// TIA Portal V17 export
// export: Created 2022-07-20T07:02:32.9247407Z, ExportSetting WithDefaults, DisplayName Totally Integrated Automation Portal, DisplayVersion V17, DisplayName TIA Portal Openness, DisplayVersion V17, DisplayName TIA Portal Version Control Interface, DisplayVersion V17, DisplayName SINAMICS Startdrive Advanced, DisplayVersion V17, DisplayName SINAMICS Startdrive G130, G150, S120, S150, SINAMICS MV, S210, DisplayVersion V17, DisplayName SINAMICS Startdrive G110M, G120, G120C, G120D, G120P, G115D, DisplayVersion V17, DisplayName STEP 7 Professional, DisplayVersion V17, DisplayName STEP 7 Safety, DisplayVersion V17, DisplayName WinCC Advanced, DisplayVersion V17
FUNCTION_BLOCK "FB11006_HeatingRegulation"   // FB11006, LAD
TITLE = Manage heating regulation
{ S7_Optimized_Access := 'TRUE' }
VERSION : 0.1
// stored: AutoNumber false, IsIECCheckEnabled false, IsRetainMemResEnabled false, MemoryReserve 100, SetENOAutomatically false, UDAEnableTagReadback false
   VAR_INPUT
      RequestInternalLampActivation { ExternalAccessible := 'False'; ExternalVisible := 'False'; ExternalWritable := 'False'} : Bool;
      SetpointTemperature { ExternalAccessible := 'False'; ExternalVisible := 'False'; ExternalWritable := 'False'} : Real;
      Reset { ExternalAccessible := 'False'; ExternalVisible := 'False'; ExternalWritable := 'False'} : Bool;
      TemperatureConfig { ExternalAccessible := 'False'; ExternalVisible := 'False'; ExternalWritable := 'False'} : "stTemperatureConfiguration";
      PIDConfig { ExternalAccessible := 'False'; ExternalVisible := 'False'; ExternalWritable := 'False'} : "stPIDConfiguration";
      TemperatureSensor : Int;
      ManualOptimisation : Bool;
   END_VAR
   VAR_OUTPUT
      ActiveHeating { ExternalAccessible := 'False'; ExternalVisible := 'False'; ExternalWritable := 'False'} : Bool;
      Error { ExternalAccessible := 'False'; ExternalVisible := 'False'; ExternalWritable := 'False'} : Bool;
      Alarm { ExternalAccessible := 'False'; ExternalVisible := 'False'; ExternalWritable := 'False'} : Bool;
      Warning { ExternalAccessible := 'False'; ExternalVisible := 'False'; ExternalWritable := 'False'} : Bool;
      SetPointOutput : Int;
   END_VAR
   VAR_IN_OUT
      Temperature : Real;
      PID : PID_Compact;
   END_VAR
   VAR
      R_TRIG_Enable : R_TRIG;
      F_TRIG_Enable { S7_SetPoint := 'True'} : F_TRIG;
      FB10022_Average_Instance { S7_SetPoint := 'True'} : "FB10022_Average";
      statDataAverage { S7_SetPoint := 'True'} : Array[0..29] of Real;
      statTemperatureAverage : Real;
      pid_state : Int;
      pid_error : Bool;
      pid_errorBits : DWord;
   END_VAR
   VAR_TEMP
      RET_VAL : Word;
   END_VAR
BEGIN

REGION Network 1 (SCL): Comments
   //==========================================================================================
   // SIEMENS SAS      RC-FR DI FA APC
   //------------------------------------------------------------------------------------------
   // Restrictions:    TIA V16 and more
   // Requirements:    S7-1500 + MGI library
   // Functionality:   This function block manage a PID regulation for temperature
   //------------------------------------------------------------------------------------------
   // Change log table:
   // Version      Date        Expert in charge    Changes applied
   // 01.00.01     09.06.2020  RTO                 First released version
   //==========================================================================================
END_REGION

REGION Network 2 (SCL): First Scan
   IF "FirstScan" THEN

       // Interface
       #ActiveHeating := FALSE;
       #SetPointOutput := 0;

       // #PID
       #PID.Mode := 0;
       #PID.ModeActivate := TRUE;
       #PID.IntegralResetMode := 1;

   END_IF;
END_REGION

REGION Network 3 (SCL): Edge Signal Management
   REGION EDGE SIGNALS
       #R_TRIG_Enable(CLK := #RequestInternalLampActivation);
       #F_TRIG_Enable(CLK := #RequestInternalLampActivation);

   END_REGION
END_REGION

REGION Network 4 (SCL): Convert analog input in temperature value
   #Temperature := #TemperatureConfig.ShiftFactor * #TemperatureSensor/10.0;
END_REGION

REGION Network 5: Average temperature over 30 secondes
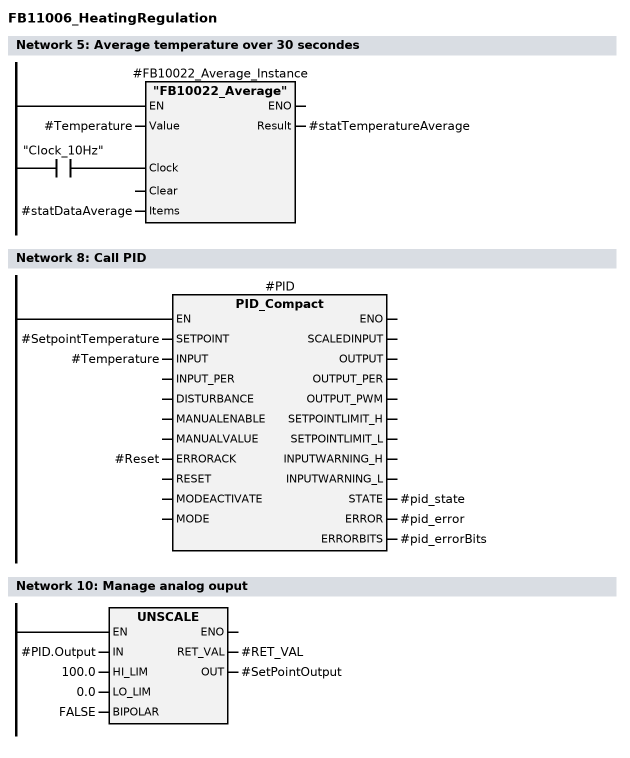
   RUNG wire#powerrail
      #FB10022_Average_Instance(Clock := wire#w1, Value := #Temperature, Clear :=, Items := #statDataAverage, Result => #statTemperatureAverage)
   END_RUNG
   RUNG wire#powerrail
      Contact( "Clock_10Hz" )
   END_RUNG wire#w1
   // the same network as SCL:
   #FB10022_Average_Instance(Value := #Temperature,   // "FB10022_Average"
                           Clock := "Clock_10Hz",
                           Items := #statDataAverage,
                           Result => #statTemperatureAverage);
END_REGION

REGION Network 6 (SCL): Manage PID
   IF NOT #ManualOptimisation THEN

       IF #R_TRIG_Enable.Q THEN
           #PID.Retain.CtrlParams.Gain := #PIDConfig.Kp;
           #PID.Retain.CtrlParams.Ti := #PIDConfig.Ki;
           #PID.Retain.CtrlParams.Td := #PIDConfig.Kd;
           #PID.Mode := 3;
           #PID.ModeActivate := TRUE;
       END_IF;

       IF #RequestInternalLampActivation THEN
           IF #PID.State = 3 AND #PID.ModeActivate THEN
               #PID.ModeActivate := FALSE;
           END_IF;
       END_IF;


       IF #F_TRIG_Enable.Q THEN
           #PID.Retain.CtrlParams.Gain := #PIDConfig.Kp;
           #PID.Retain.CtrlParams.Ti := #PIDConfig.Ki;
           #PID.Retain.CtrlParams.Td := #PIDConfig.Kd;
           #PID.Mode := 0;
           #PID.ModeActivate := TRUE;
       END_IF;

       IF NOT #RequestInternalLampActivation THEN
           IF #PID.State = 0 AND #PID.ModeActivate THEN
               #PID.ModeActivate := FALSE;
           END_IF;
       END_IF;

   END_IF;
END_REGION

REGION Network 7 (SCL): Reset PID if disabled
   #PID.Reset := (#Reset OR (#pid_state = 0 AND #RequestInternalLampActivation))AND NOT #PID.Reset;
END_REGION

REGION Network 8: Call PID
   RUNG wire#powerrail
      #PID.PID_Compact(Setpoint := #SetpointTemperature, Input := #Temperature, Input_PER :=, Disturbance :=, ManualEnable :=, ManualValue :=, ErrorAck := #Reset, Reset :=, ModeActivate :=, Mode :=, ScaledInput =>, Output =>, Output_PER =>, Output_PWM =>, SetpointLimit_H =>, SetpointLimit_L =>, InputWarning_H =>, InputWarning_L =>, State => #pid_state, Error => #pid_error, ErrorBits => #pid_errorBits)
   END_RUNG
   // the same network as SCL:
   #PID(Setpoint := #SetpointTemperature,   // PID_Compact
        Input := #Temperature,
        ErrorAck := #Reset,
        State => #pid_state,
        Error => #pid_error,
        ErrorBits => #pid_errorBits);
END_REGION

REGION Network 9 (SCL): Manage Output
   #Error := #PID.Error;//OR #statTemperatureAverage > #TemperatureConfig.AlarmWindow;
   #ActiveHeating := #RequestInternalLampActivation AND NOT #Error;
END_REGION

REGION Network 10: Manage analog ouput
   RUNG wire#powerrail
      UNSCALE(IN := #PID.Output, HI_LIM := 100.0, LO_LIM := 0.0, BIPOLAR := FALSE, RET_VAL => #RET_VAL, OUT => #SetPointOutput)
   END_RUNG
   // the same network as SCL:
   #RET_VAL := UNSCALE(IN := #PID.Output,
                       HI_LIM := 100.0,
                       LO_LIM := 0.0,
                       BIPOLAR := FALSE,
                       OUT => #SetPointOutput);
END_REGION

REGION Network 11 (SCL): Manage Warning and Alarm on temperature
   //IF #RequestInternalLampActivation THEN


       IF ABS(#SetpointTemperature - #Temperature) > #TemperatureConfig.AlarmWindow THEN
           #Alarm := TRUE;
           #Warning := FALSE;
           ELSIF ABS(#SetpointTemperature - #Temperature) > #TemperatureConfig.WarningWindow THEN
               #Warning := TRUE;
               #Alarm := FALSE;
           ELSE
               #Warning := FALSE;
               #Alarm := FALSE;
           END_IF;
   //    END_IF;


   IF NOT #ActiveHeating THEN
       #SetPointOutput := 0;
   END_IF;


   IF #Reset THEN
       #Warning := FALSE;
       #Alarm := FALSE;
   END_IF;
END_REGION
END_FUNCTION_BLOCK
